// Mitsubishi GX Works2 project: PLC 미니 프로젝트   PLC: Q03UDV

PROGRAM MAIN
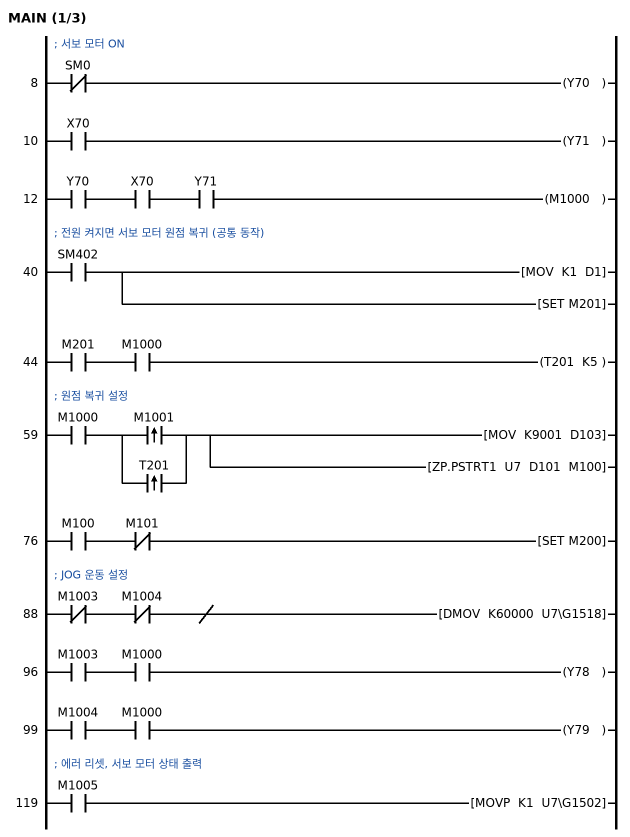
; 서보 모터 ON
8     LDI     SM0
      OUT     Y70
10    LD      X70
      OUT     Y71
12    LD      Y70
      AND     X70
      AND     Y71
      OUT     M1000
; 전원 켜지면 서보 모터 원점 복귀 (공통 동작)
40    LD      SM402
      MOV     K1 D1
      SET     M201
44    LD      M201
      AND     M1000
      OUT     T201 K5
; 원점 복귀 설정
59    LD      M1000
      LDP     M1001
      ORP     T201
      ANB
      MOV     K9001 D103
      ZP.PSTRT1 U7 D101 M100
76    LD      M100
      ANI     M101
      SET     M200
; JOG 운동 설정
88    LDI     M1003
      ANI     M1004
      INV
      DMOV    K60000 U7\G1518
96    LD      M1003
      AND     M1000
      OUT     Y78
99    LD      M1004
      AND     M1000
      OUT     Y79
; 에러 리셋, 서보 모터 상태 출력
119   LD      M1005
      MOVP    K1 U7\G1502
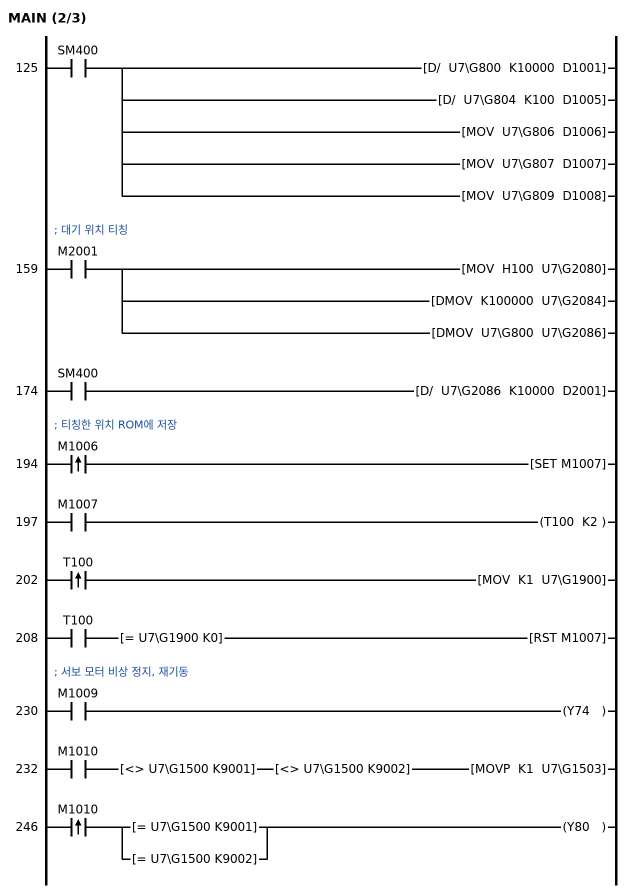
125   LD      SM400
      D/      U7\G800 K10000 D1001
      D/      U7\G804 K100 D1005
      MOV     U7\G806 D1006
      MOV     U7\G807 D1007
      MOV     U7\G809 D1008
; 대기 위치 티칭
159   LD      M2001
      MOV     H100 U7\G2080
      DMOV    K100000 U7\G2084
      DMOV    U7\G800 U7\G2086
174   LD      SM400
      D/      U7\G2086 K10000 D2001
; 티칭한 위치 ROM에 저장
194   LDP     M1006
      SET     M1007
197   LD      M1007
      OUT     T100 K2
202   LDP     T100
      MOV     K1 U7\G1900
208   LD      T100
      AND=    U7\G1900 K0
      RST     M1007
; 서보 모터 비상 정지, 재기동
230   LD      M1009
      OUT     Y74
232   LD      M1010
      AND<>   U7\G1500 K9001
      AND<>   U7\G1500 K9002
      MOVP    K1 U7\G1503
246   LDP     M1010
      LD=     U7\G1500 K9001
      OR=     U7\G1500 K9002
      ANB
      OUT     Y80
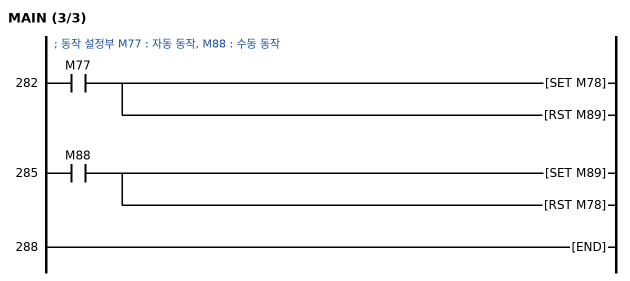
; 동작 설정부 M77 : 자동 동작, M88 : 수동 동작
282   LD      M77
      SET     M78
      RST     M89
285   LD      M88
      SET     M89
      RST     M78
288   END
END_PROGRAM

PROGRAM FacCheck
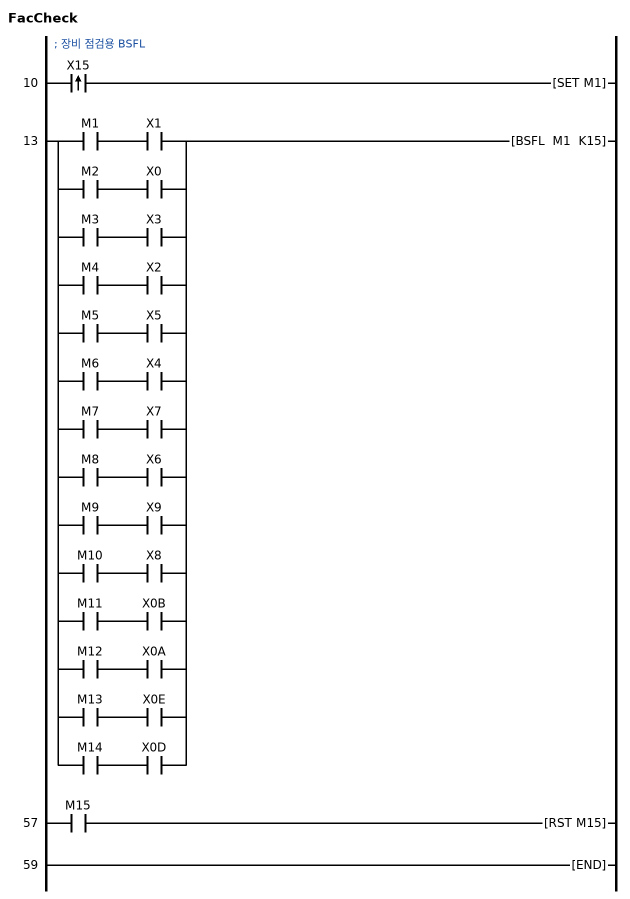
; 장비 점검용 BSFL
10    LDP     X15
      SET     M1
13    LD      M1
      AND     X1
      LD      M2
      AND     X0
      ORB
      LD      M3
      AND     X3
      ORB
      LD      M4
      AND     X2
      ORB
      LD      M5
      AND     X5
      ORB
      LD      M6
      AND     X4
      ORB
      LD      M7
      AND     X7
      ORB
      LD      M8
      AND     X6
      ORB
      LD      M9
      AND     X9
      ORB
      LD      M10
      AND     X8
      ORB
      LD      M11
      AND     X0B
      ORB
      LD      M12
      AND     X0A
      ORB
      LD      M13
      AND     X0E
      ORB
      LD      M14
      AND     X0D
      ORB
      BSFL    M1 K15
57    LD      M15
      RST     M15
59    END
END_PROGRAM

PROGRAM Auto
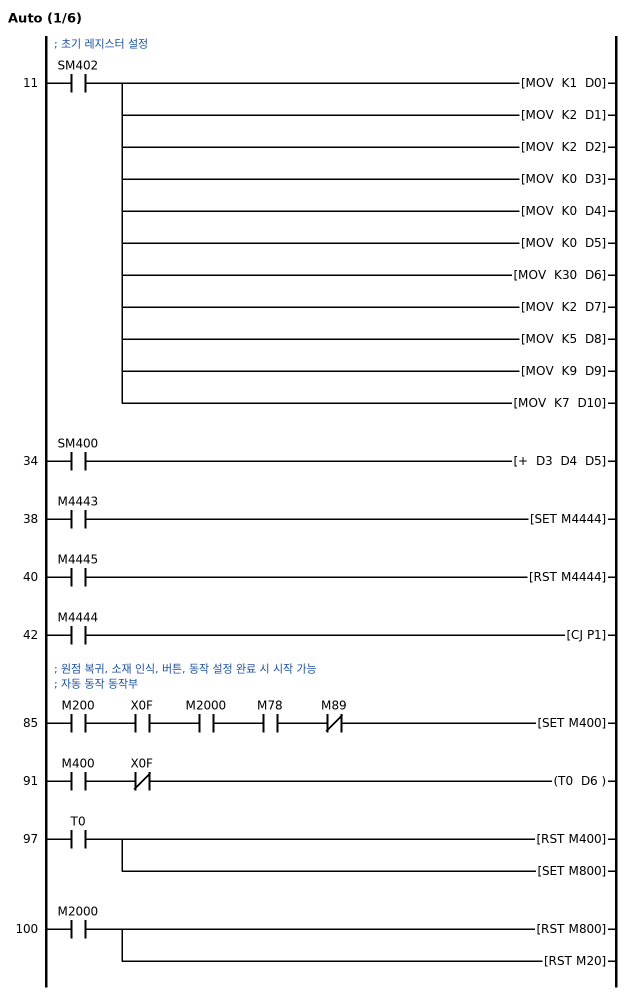
; 초기 레지스터 설정
11    LD      SM402
      MOV     K1 D0
      MOV     K2 D1
      MOV     K2 D2
      MOV     K0 D3
      MOV     K0 D4
      MOV     K0 D5
      MOV     K30 D6
      MOV     K2 D7
      MOV     K5 D8
      MOV     K9 D9
      MOV     K7 D10
34    LD      SM400
      +       D3 D4 D5
38    LD      M4443
      SET     M4444
40    LD      M4445
      RST     M4444
42    LD      M4444
      CJ      P1
; 원점 복귀, 소재 인식, 버튼, 동작 설정 완료 시 시작 가능
; 자동 동작 동작부
85    LD      M200
      AND     X0F
      AND     M2000
      AND     M78
      ANI     M89
      SET     M400
91    LD      M400
      ANI     X0F
      OUT     T0 D6
97    LD      T0
      RST     M400
      SET     M800
100   LD      M2000
      RST     M800
      RST     M20
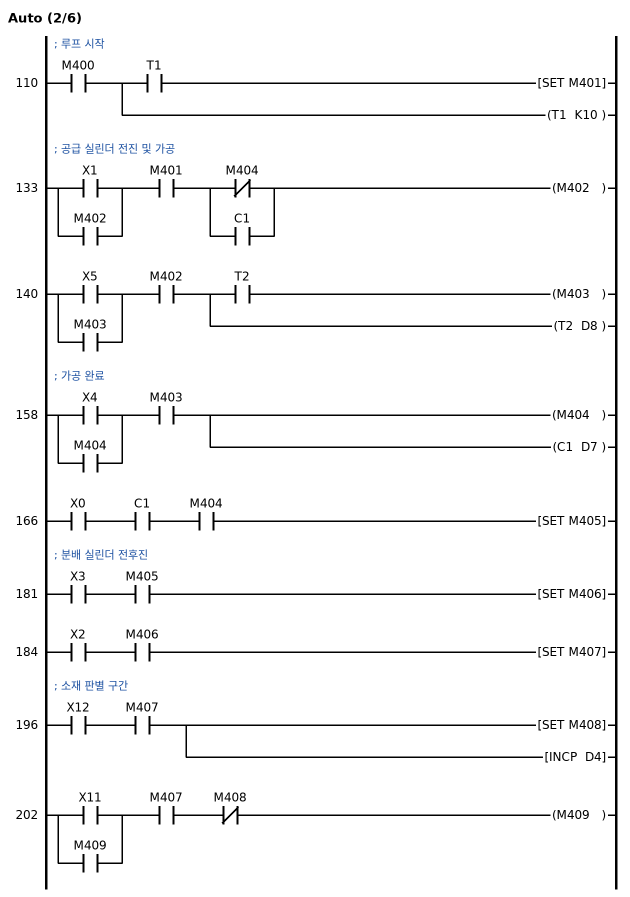
; 루프 시작
110   LD      M400
      MPS
      AND     T1
      SET     M401
      MPP
      OUT     T1 K10
; 공급 실린더 전진 및 가공
133   LD      X1
      OR      M402
      AND     M401
      LDI     M404
      OR      C1
      ANB
      OUT     M402
140   LD      X5
      OR      M403
      AND     M402
      MPS
      AND     T2
      OUT     M403
      MPP
      OUT     T2 D8
; 가공 완료
158   LD      X4
      OR      M404
      AND     M403
      OUT     M404
      OUT     C1 D7
166   LD      X0
      AND     C1
      AND     M404
      SET     M405
; 분배 실린더 전후진
181   LD      X3
      AND     M405
      SET     M406
184   LD      X2
      AND     M406
      SET     M407
; 소재 판별 구간
196   LD      X12
      AND     M407
      SET     M408
      INCP    D4
202   LD      X11
      OR      M409
      AND     M407
      ANI     M408
      OUT     M409
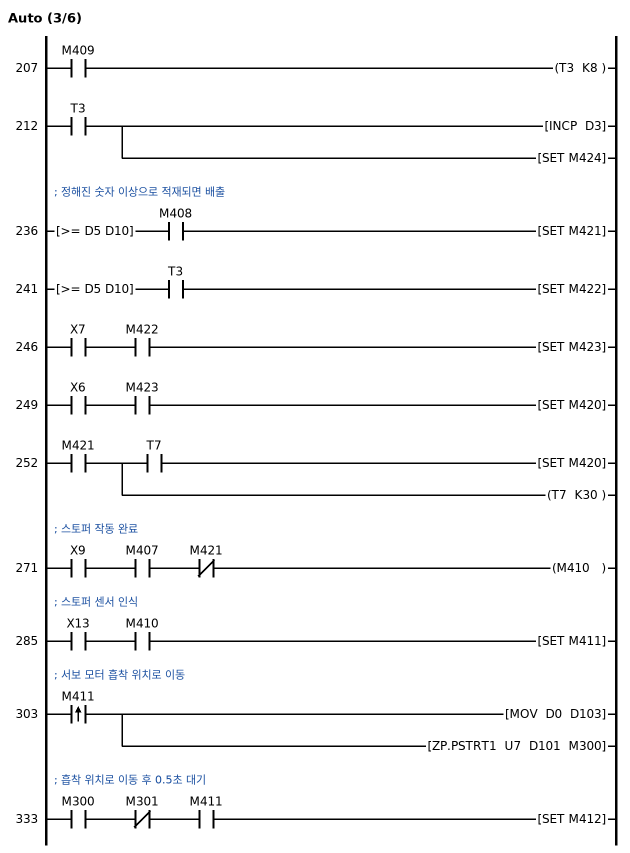
207   LD      M409
      OUT     T3 K8
212   LD      T3
      INCP    D3
      SET     M424
; 정해진 숫자 이상으로 적재되면 배출
236   LD>=    D5 D10
      AND     M408
      SET     M421
241   LD>=    D5 D10
      AND     T3
      SET     M422
246   LD      X7
      AND     M422
      SET     M423
249   LD      X6
      AND     M423
      SET     M420
252   LD      M421
      MPS
      AND     T7
      SET     M420
      MPP
      OUT     T7 K30
; 스토퍼 작동 완료
271   LD      X9
      AND     M407
      ANI     M421
      OUT     M410
; 스토퍼 센서 인식
285   LD      X13
      AND     M410
      SET     M411
; 서보 모터 흡착 위치로 이동
303   LDP     M411
      MOV     D0 D103
      ZP.PSTRT1 U7 D101 M300
; 흡착 위치로 이동 후 0.5초 대기
333   LD      M300
      ANI     M301
      AND     M411
      SET     M412
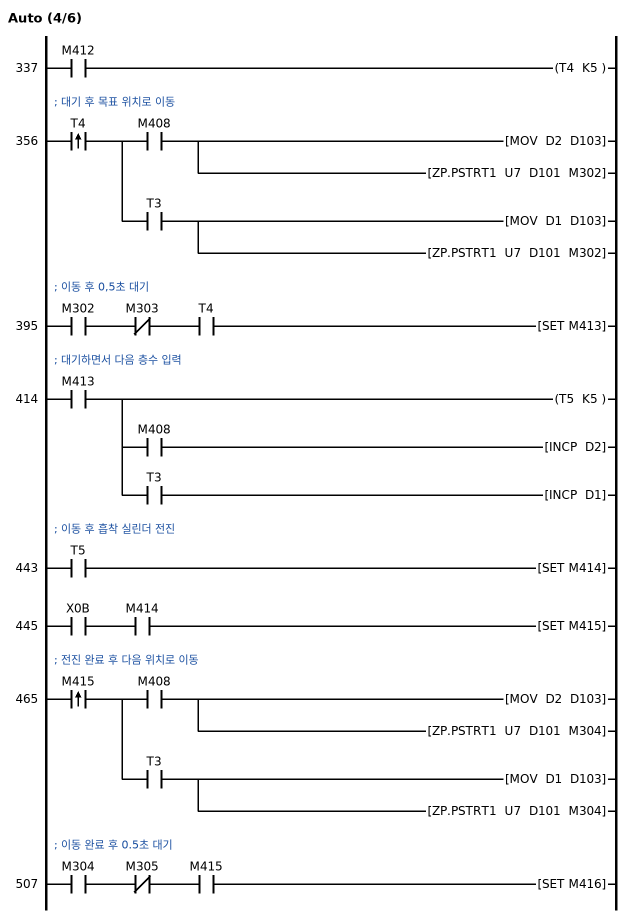
337   LD      M412
      OUT     T4 K5
; 대기 후 목표 위치로 이동
356   LDP     T4
      MPS
      AND     M408
      MOV     D2 D103
      ZP.PSTRT1 U7 D101 M302
      MPP
      AND     T3
      MOV     D1 D103
      ZP.PSTRT1 U7 D101 M302
; 이동 후 0,5초 대기
395   LD      M302
      ANI     M303
      AND     T4
      SET     M413
; 대기하면서 다음 층수 입력
414   LD      M413
      OUT     T5 K5
      MPS
      AND     M408
      INCP    D2
      MPP
      AND     T3
      INCP    D1
; 이동 후 흡착 실린더 전진
443   LD      T5
      SET     M414
445   LD      X0B
      AND     M414
      SET     M415
; 전진 완료 후 다음 위치로 이동
465   LDP     M415
      MPS
      AND     M408
      MOV     D2 D103
      ZP.PSTRT1 U7 D101 M304
      MPP
      AND     T3
      MOV     D1 D103
      ZP.PSTRT1 U7 D101 M304
; 이동 완료 후 0.5초 대기
507   LD      M304
      ANI     M305
      AND     M415
      SET     M416
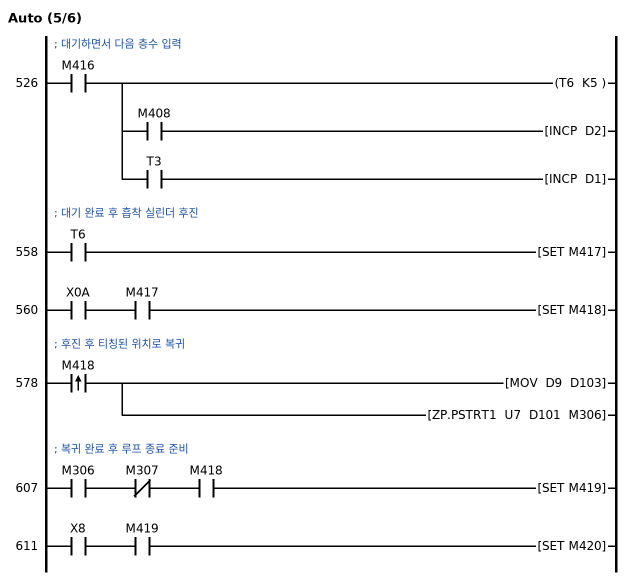
; 대기하면서 다음 층수 입력
526   LD      M416
      OUT     T6 K5
      MPS
      AND     M408
      INCP    D2
      MPP
      AND     T3
      INCP    D1
; 대기 완료 후 흡착 실린더 후진
558   LD      T6
      SET     M417
560   LD      X0A
      AND     M417
      SET     M418
; 후진 후 티칭된 위치로 복귀
578   LDP     M418
      MOV     D9 D103
      ZP.PSTRT1 U7 D101 M306
; 복귀 완료 후 루프 종료 준비
607   LD      M306
      ANI     M307
      AND     M418
      SET     M419
611   LD      X8
      AND     M419
      SET     M420
      P1
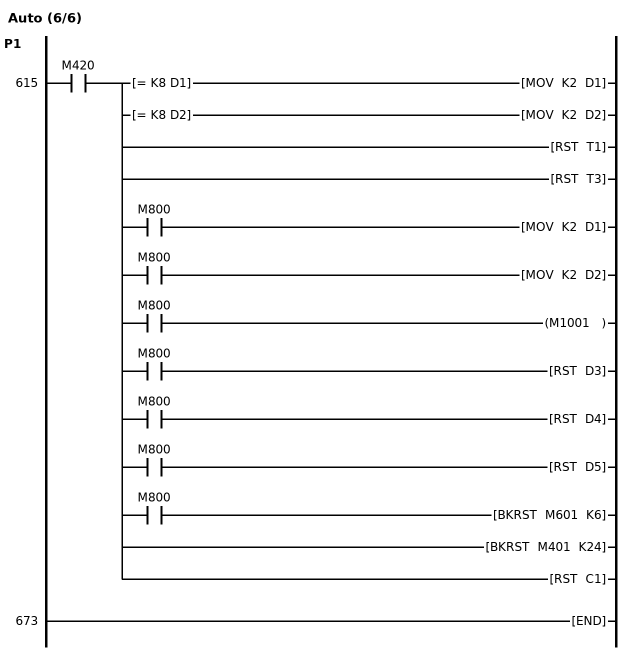
615   LD      M420
      MPS
      AND=    K8 D1
      MOV     K2 D1
      MRD
      AND=    K8 D2
      MOV     K2 D2
      MPP
      RST     T1
      RST     T3
      MPS
      AND     M800
      MOV     K2 D1
      MRD
      AND     M800
      MOV     K2 D2
      MRD
      AND     M800
      OUT     M1001
      MRD
      AND     M800
      RST     D3
      MRD
      AND     M800
      RST     D4
      MRD
      AND     M800
      RST     D5
      MRD
      AND     M800
      BKRST   M601 K6
      MPP
      BKRST   M401 K24
      RST     C1
673   END
END_PROGRAM

PROGRAM Output
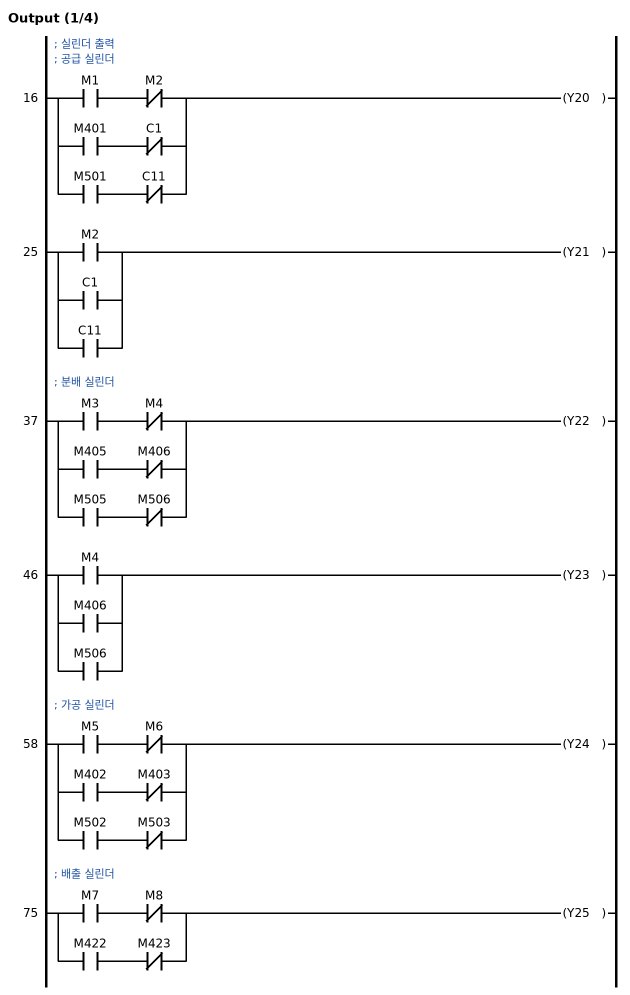
; 실린더 출력
; 공급 실린더
16    LD      M1
      ANI     M2
      LD      M401
      ANI     C1
      ORB
      LD      M501
      ANI     C11
      ORB
      OUT     Y20
25    LD      M2
      OR      C1
      OR      C11
      OUT     Y21
; 분배 실린더
37    LD      M3
      ANI     M4
      LD      M405
      ANI     M406
      ORB
      LD      M505
      ANI     M506
      ORB
      OUT     Y22
46    LD      M4
      OR      M406
      OR      M506
      OUT     Y23
; 가공 실린더
58    LD      M5
      ANI     M6
      LD      M402
      ANI     M403
      ORB
      LD      M502
      ANI     M503
      ORB
      OUT     Y24
; 배출 실린더
75    LD      M7
      ANI     M8
      LD      M422
      ANI     M423
      ORB
      OUT     Y25
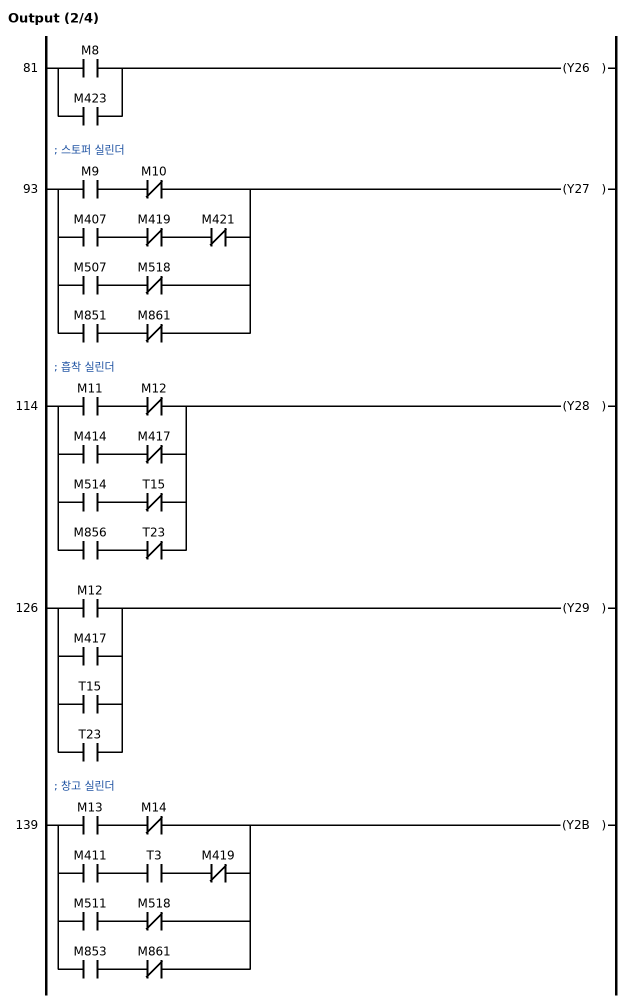
81    LD      M8
      OR      M423
      OUT     Y26
; 스토퍼 실린더
93    LD      M9
      ANI     M10
      LD      M407
      ANI     M419
      ANI     M421
      ORB
      LD      M507
      ANI     M518
      ORB
      LD      M851
      ANI     M861
      ORB
      OUT     Y27
; 흡착 실린더
114   LD      M11
      ANI     M12
      LD      M414
      ANI     M417
      ORB
      LD      M514
      ANI     T15
      ORB
      LD      M856
      ANI     T23
      ORB
      OUT     Y28
126   LD      M12
      OR      M417
      OR      T15
      OR      T23
      OUT     Y29
; 창고 실린더
139   LD      M13
      ANI     M14
      LD      M411
      AND     T3
      ANI     M419
      ORB
      LD      M511
      ANI     M518
      ORB
      LD      M853
      ANI     M861
      ORB
      OUT     Y2B
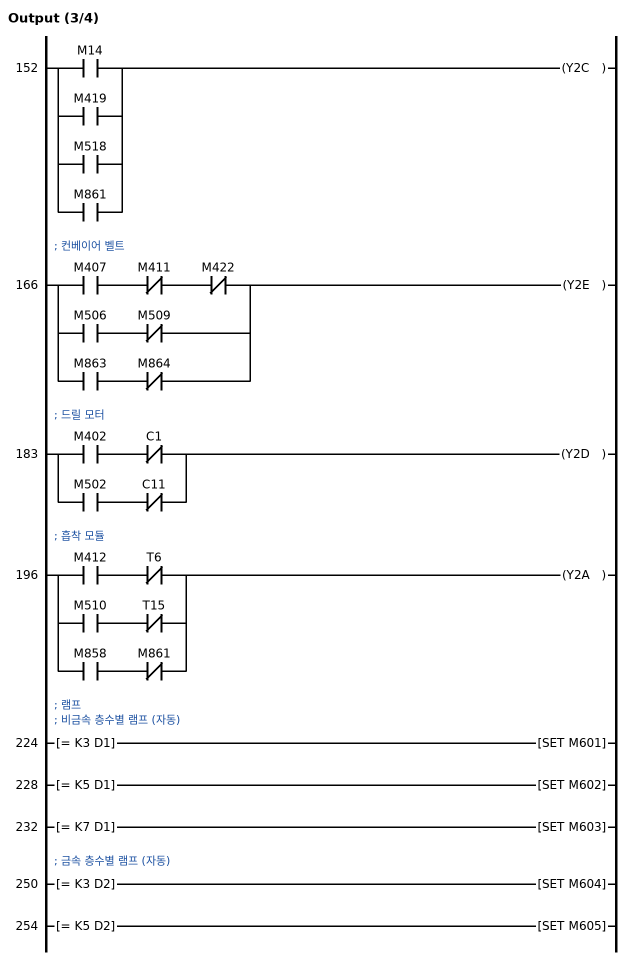
152   LD      M14
      OR      M419
      OR      M518
      OR      M861
      OUT     Y2C
; 컨베이어 벨트
166   LD      M407
      ANI     M411
      ANI     M422
      LD      M506
      ANI     M509
      ORB
      LD      M863
      ANI     M864
      ORB
      OUT     Y2E
; 드릴 모터
183   LD      M402
      ANI     C1
      LD      M502
      ANI     C11
      ORB
      OUT     Y2D
; 흡착 모듈
196   LD      M412
      ANI     T6
      LD      M510
      ANI     T15
      ORB
      LD      M858
      ANI     M861
      ORB
      OUT     Y2A
; 램프
; 비금속 층수별 램프 (자동)
224   LD=     K3 D1
      SET     M601
228   LD=     K5 D1
      SET     M602
232   LD=     K7 D1
      SET     M603
; 금속 층수별 램프 (자동)
250   LD=     K3 D2
      SET     M604
254   LD=     K5 D2
      SET     M605
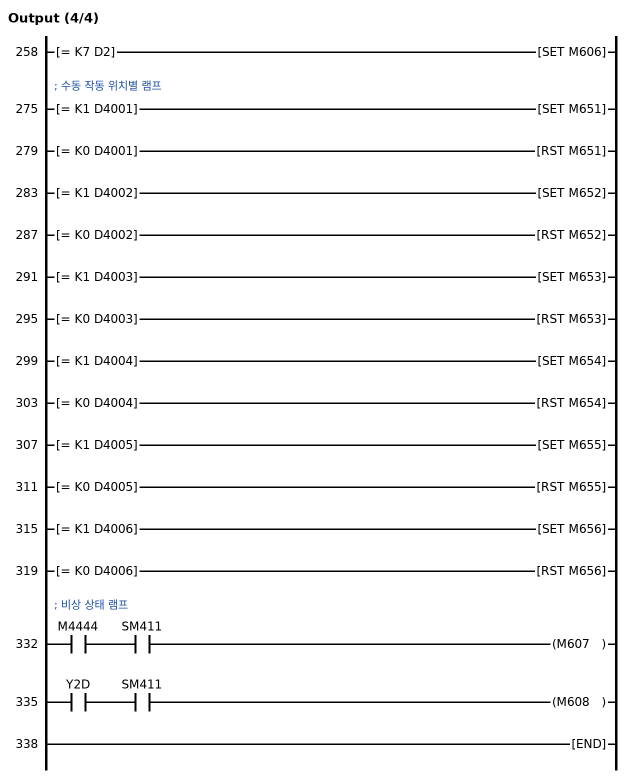
258   LD=     K7 D2
      SET     M606
; 수동 작동 위치별 램프
275   LD=     K1 D4001
      SET     M651
279   LD=     K0 D4001
      RST     M651
283   LD=     K1 D4002
      SET     M652
287   LD=     K0 D4002
      RST     M652
291   LD=     K1 D4003
      SET     M653
295   LD=     K0 D4003
      RST     M653
299   LD=     K1 D4004
      SET     M654
303   LD=     K0 D4004
      RST     M654
307   LD=     K1 D4005
      SET     M655
311   LD=     K0 D4005
      RST     M655
315   LD=     K1 D4006
      SET     M656
319   LD=     K0 D4006
      RST     M656
; 비상 상태 램프
332   LD      M4444
      AND     SM411
      OUT     M607
335   LD      Y2D
      AND     SM411
      OUT     M608
338   END
END_PROGRAM

PROGRAM Manual
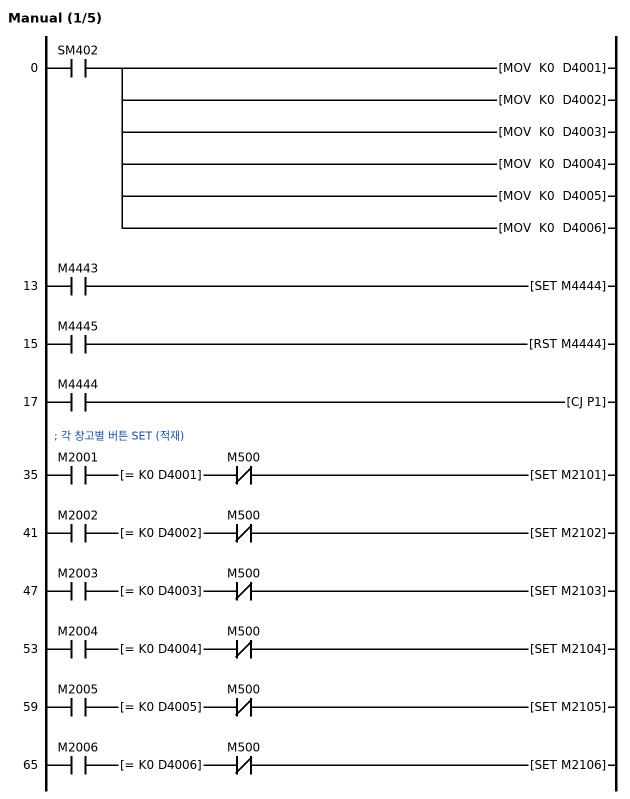
0     LD      SM402
      MOV     K0 D4001
      MOV     K0 D4002
      MOV     K0 D4003
      MOV     K0 D4004
      MOV     K0 D4005
      MOV     K0 D4006
13    LD      M4443
      SET     M4444
15    LD      M4445
      RST     M4444
17    LD      M4444
      CJ      P1
; 각 창고별 버튼 SET (적재)
35    LD      M2001
      AND=    K0 D4001
      ANI     M500
      SET     M2101
41    LD      M2002
      AND=    K0 D4002
      ANI     M500
      SET     M2102
47    LD      M2003
      AND=    K0 D4003
      ANI     M500
      SET     M2103
53    LD      M2004
      AND=    K0 D4004
      ANI     M500
      SET     M2104
59    LD      M2005
      AND=    K0 D4005
      ANI     M500
      SET     M2105
65    LD      M2006
      AND=    K0 D4006
      ANI     M500
      SET     M2106
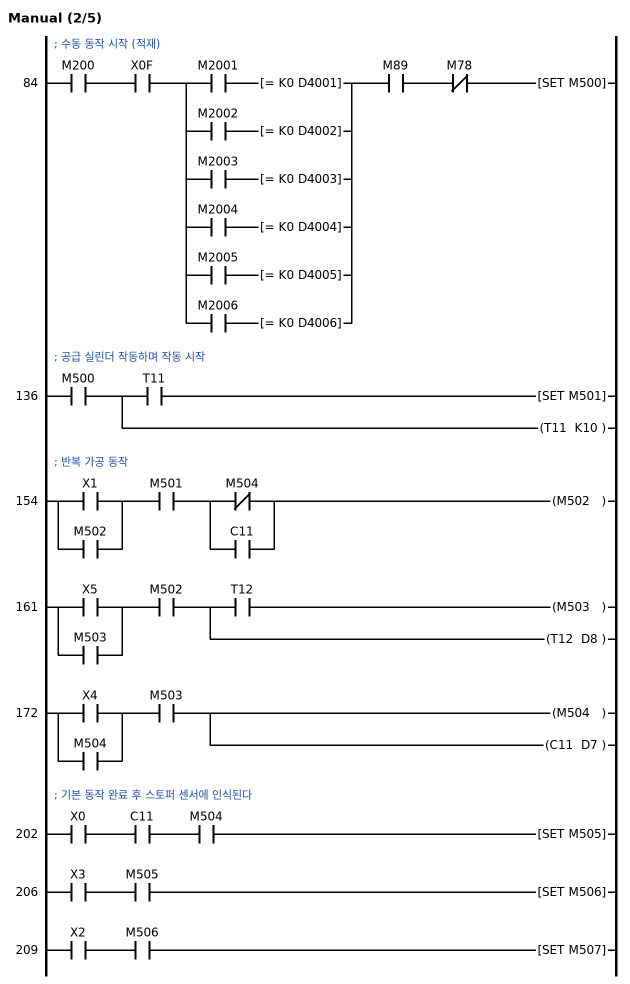
; 수동 동작 시작 (적재)
84    LD      M200
      AND     X0F
      LD      M2001
      AND=    K0 D4001
      LD      M2002
      AND=    K0 D4002
      ORB
      LD      M2003
      AND=    K0 D4003
      ORB
      LD      M2004
      AND=    K0 D4004
      ORB
      LD      M2005
      AND=    K0 D4005
      ORB
      LD      M2006
      AND=    K0 D4006
      ORB
      ANB
      AND     M89
      ANI     M78
      SET     M500
; 공급 실린더 작동하며 작동 시작
136   LD      M500
      MPS
      AND     T11
      SET     M501
      MPP
      OUT     T11 K10
; 반복 가공 동작
154   LD      X1
      OR      M502
      AND     M501
      LDI     M504
      OR      C11
      ANB
      OUT     M502
161   LD      X5
      OR      M503
      AND     M502
      MPS
      AND     T12
      OUT     M503
      MPP
      OUT     T12 D8
172   LD      X4
      OR      M504
      AND     M503
      OUT     M504
      OUT     C11 D7
; 기본 동작 완료 후 스토퍼 센서에 인식된다
202   LD      X0
      AND     C11
      AND     M504
      SET     M505
206   LD      X3
      AND     M505
      SET     M506
209   LD      X2
      AND     M506
      SET     M507
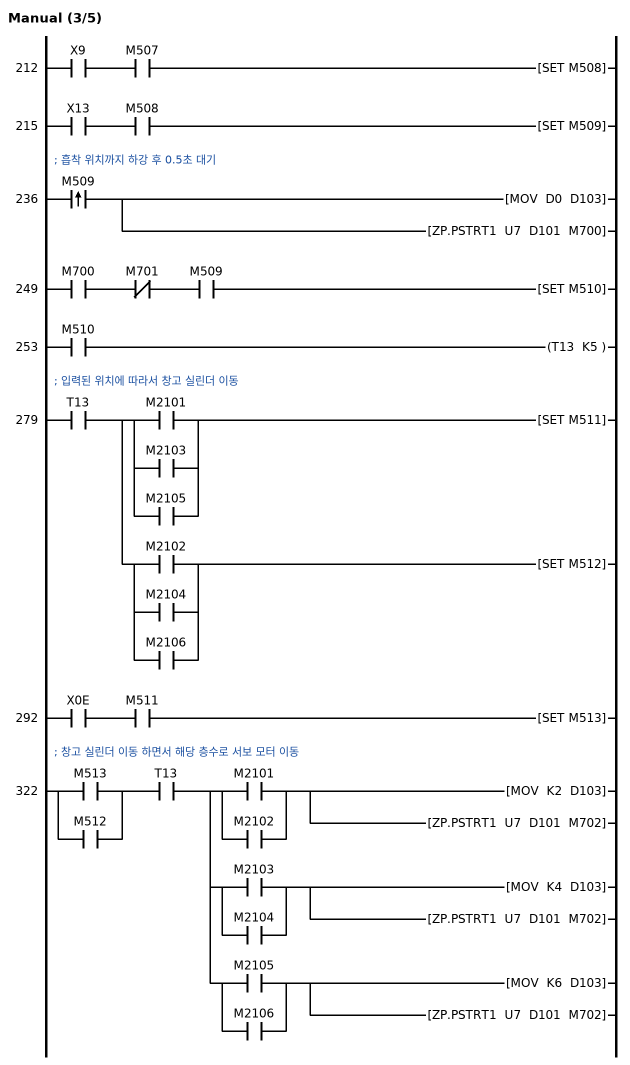
212   LD      X9
      AND     M507
      SET     M508
215   LD      X13
      AND     M508
      SET     M509
; 흡착 위치까지 하강 후 0.5초 대기
236   LDP     M509
      MOV     D0 D103
      ZP.PSTRT1 U7 D101 M700
249   LD      M700
      ANI     M701
      AND     M509
      SET     M510
253   LD      M510
      OUT     T13 K5
; 입력된 위치에 따라서 창고 실린더 이동
279   LD      T13
      MPS
      LD      M2101
      OR      M2103
      OR      M2105
      ANB
      SET     M511
      MPP
      LD      M2102
      OR      M2104
      OR      M2106
      ANB
      SET     M512
292   LD      X0E
      AND     M511
      SET     M513
; 창고 실린더 이동 하면서 해당 층수로 서보 모터 이동
322   LD      M513
      OR      M512
      AND     T13
      MPS
      LD      M2101
      OR      M2102
      ANB
      MOV     K2 D103
      ZP.PSTRT1 U7 D101 M702
      MRD
      LD      M2103
      OR      M2104
      ANB
      MOV     K4 D103
      ZP.PSTRT1 U7 D101 M702
      MPP
      LD      M2105
      OR      M2106
      ANB
      MOV     K6 D103
      ZP.PSTRT1 U7 D101 M702
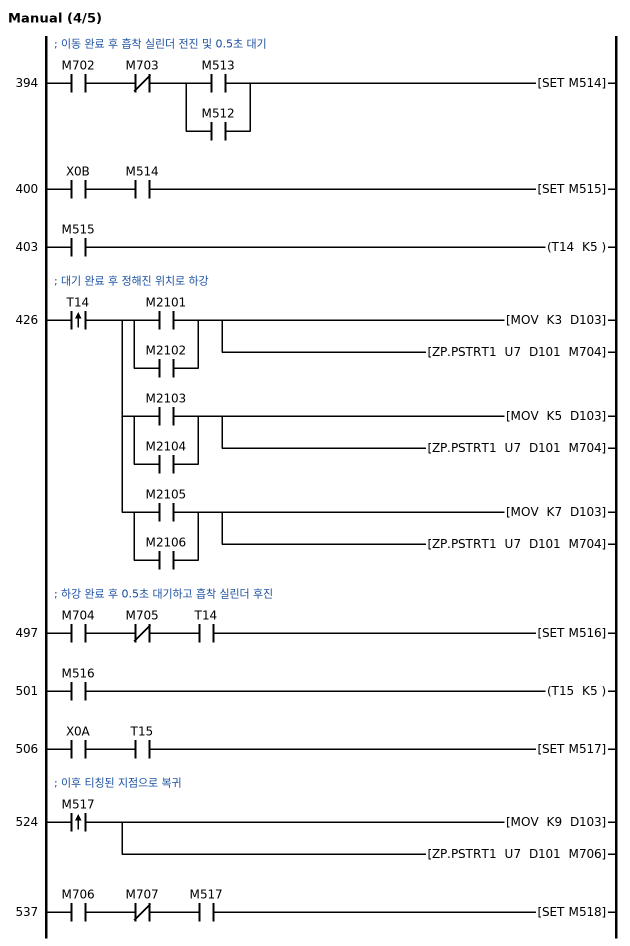
; 이동 완료 후 흡착 실린더 전진 및 0.5초 대기
394   LD      M702
      ANI     M703
      LD      M513
      OR      M512
      ANB
      SET     M514
400   LD      X0B
      AND     M514
      SET     M515
403   LD      M515
      OUT     T14 K5
; 대기 완료 후 정해진 위치로 하강
426   LDP     T14
      MPS
      LD      M2101
      OR      M2102
      ANB
      MOV     K3 D103
      ZP.PSTRT1 U7 D101 M704
      MRD
      LD      M2103
      OR      M2104
      ANB
      MOV     K5 D103
      ZP.PSTRT1 U7 D101 M704
      MPP
      LD      M2105
      OR      M2106
      ANB
      MOV     K7 D103
      ZP.PSTRT1 U7 D101 M704
; 하강 완료 후 0.5초 대기하고 흡착 실린더 후진
497   LD      M704
      ANI     M705
      AND     T14
      SET     M516
501   LD      M516
      OUT     T15 K5
506   LD      X0A
      AND     T15
      SET     M517
; 이후 티칭된 지점으로 복귀
524   LDP     M517
      MOV     K9 D103
      ZP.PSTRT1 U7 D101 M706
537   LD      M706
      ANI     M707
      AND     M517
      SET     M518
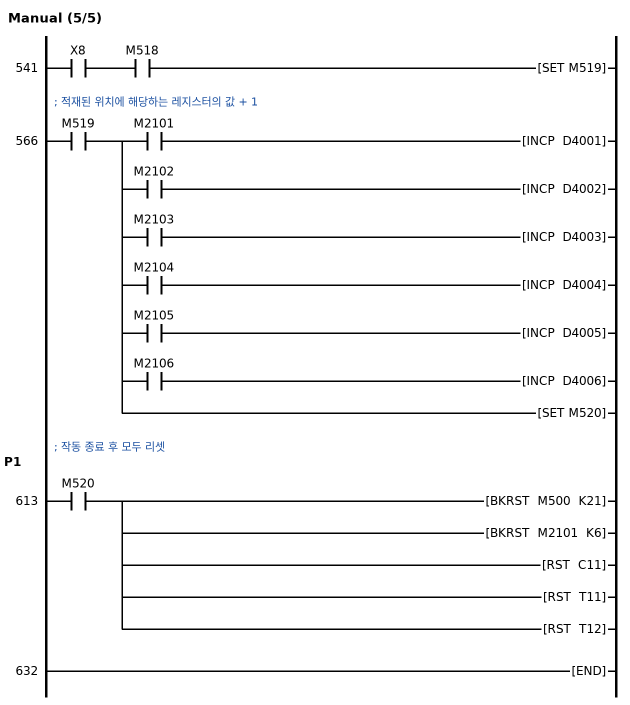
541   LD      X8
      AND     M518
      SET     M519
; 적재된 위치에 해당하는 레지스터의 값 + 1
566   LD      M519
      MPS
      AND     M2101
      INCP    D4001
      MRD
      AND     M2102
      INCP    D4002
      MRD
      AND     M2103
      INCP    D4003
      MRD
      AND     M2104
      INCP    D4004
      MRD
      AND     M2105
      INCP    D4005
      MRD
      AND     M2106
      INCP    D4006
      MPP
      SET     M520
; 작동 종료 후 모두 리셋
      P1
613   LD      M520
      BKRST   M500 K21
      BKRST   M2101 K6
      RST     C11
      RST     T11
      RST     T12
632   END
END_PROGRAM

PROGRAM Manual_2
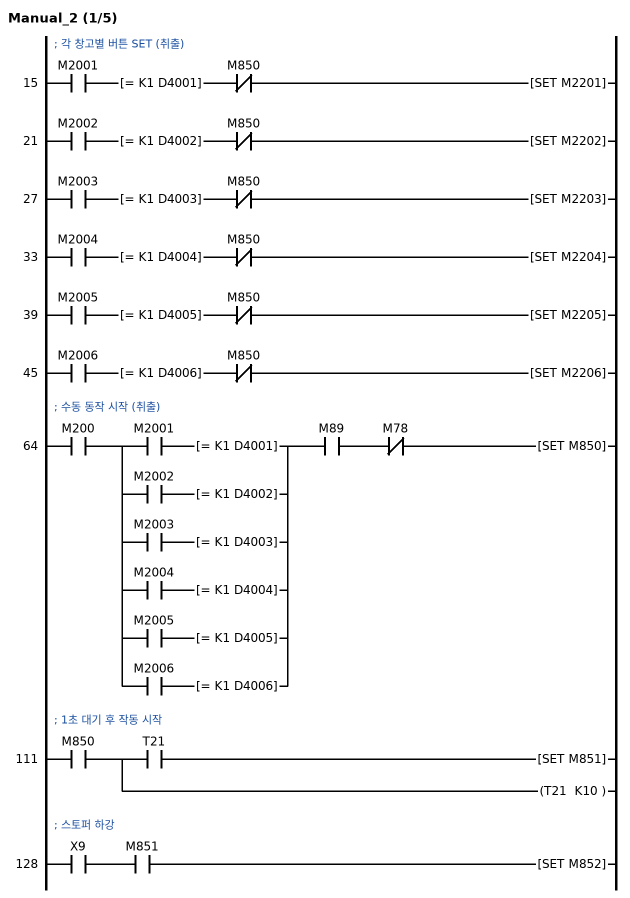
; 각 창고별 버튼 SET (취출)
15    LD      M2001
      AND=    K1 D4001
      ANI     M850
      SET     M2201
21    LD      M2002
      AND=    K1 D4002
      ANI     M850
      SET     M2202
27    LD      M2003
      AND=    K1 D4003
      ANI     M850
      SET     M2203
33    LD      M2004
      AND=    K1 D4004
      ANI     M850
      SET     M2204
39    LD      M2005
      AND=    K1 D4005
      ANI     M850
      SET     M2205
45    LD      M2006
      AND=    K1 D4006
      ANI     M850
      SET     M2206
; 수동 동작 시작 (취출)
64    LD      M200
      LD      M2001
      AND=    K1 D4001
      LD      M2002
      AND=    K1 D4002
      ORB
      LD      M2003
      AND=    K1 D4003
      ORB
      LD      M2004
      AND=    K1 D4004
      ORB
      LD      M2005
      AND=    K1 D4005
      ORB
      LD      M2006
      AND=    K1 D4006
      ORB
      ANB
      AND     M89
      ANI     M78
      SET     M850
; 1초 대기 후 작동 시작
111   LD      M850
      MPS
      AND     T21
      SET     M851
      MPP
      OUT     T21 K10
; 스토퍼 하강
128   LD      X9
      AND     M851
      SET     M852
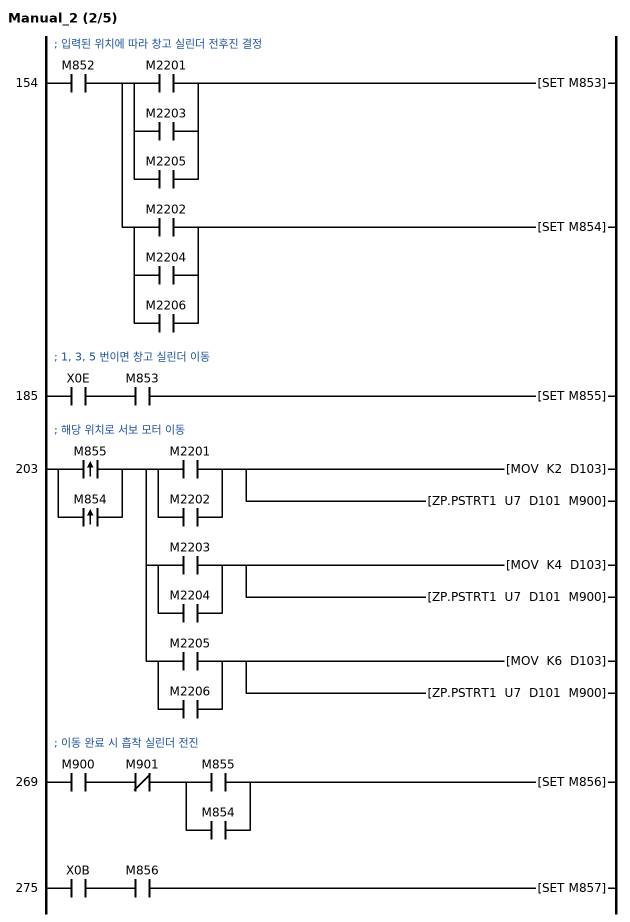
; 입력된 위치에 따라 창고 실린더 전후진 결정
154   LD      M852
      MPS
      LD      M2201
      OR      M2203
      OR      M2205
      ANB
      SET     M853
      MPP
      LD      M2202
      OR      M2204
      OR      M2206
      ANB
      SET     M854
; 1, 3, 5 번이면 창고 실린더 이동
185   LD      X0E
      AND     M853
      SET     M855
; 해당 위치로 서보 모터 이동
203   LDP     M855
      ORP     M854
      MPS
      LD      M2201
      OR      M2202
      ANB
      MOV     K2 D103
      ZP.PSTRT1 U7 D101 M900
      MRD
      LD      M2203
      OR      M2204
      ANB
      MOV     K4 D103
      ZP.PSTRT1 U7 D101 M900
      MPP
      LD      M2205
      OR      M2206
      ANB
      MOV     K6 D103
      ZP.PSTRT1 U7 D101 M900
; 이동 완료 시 흡착 실린더 전진
269   LD      M900
      ANI     M901
      LD      M855
      OR      M854
      ANB
      SET     M856
275   LD      X0B
      AND     M856
      SET     M857
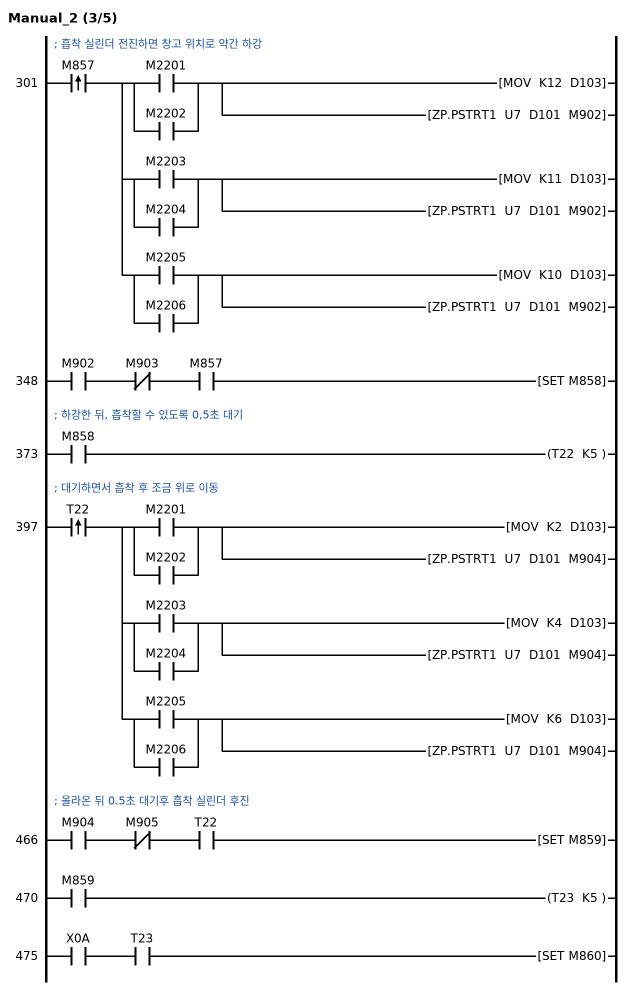
; 흡착 실린더 전진하면 창고 위치로 약간 하강
301   LDP     M857
      MPS
      LD      M2201
      OR      M2202
      ANB
      MOV     K12 D103
      ZP.PSTRT1 U7 D101 M902
      MRD
      LD      M2203
      OR      M2204
      ANB
      MOV     K11 D103
      ZP.PSTRT1 U7 D101 M902
      MPP
      LD      M2205
      OR      M2206
      ANB
      MOV     K10 D103
      ZP.PSTRT1 U7 D101 M902
348   LD      M902
      ANI     M903
      AND     M857
      SET     M858
; 하강한 뒤, 흡착할 수 있도록 0,5초 대기
373   LD      M858
      OUT     T22 K5
; 대기하면서 흡착 후 조금 위로 이동
397   LDP     T22
      MPS
      LD      M2201
      OR      M2202
      ANB
      MOV     K2 D103
      ZP.PSTRT1 U7 D101 M904
      MRD
      LD      M2203
      OR      M2204
      ANB
      MOV     K4 D103
      ZP.PSTRT1 U7 D101 M904
      MPP
      LD      M2205
      OR      M2206
      ANB
      MOV     K6 D103
      ZP.PSTRT1 U7 D101 M904
; 올라온 뒤 0.5초 대기후 흡착 실린더 후진
466   LD      M904
      ANI     M905
      AND     T22
      SET     M859
470   LD      M859
      OUT     T23 K5
475   LD      X0A
      AND     T23
      SET     M860
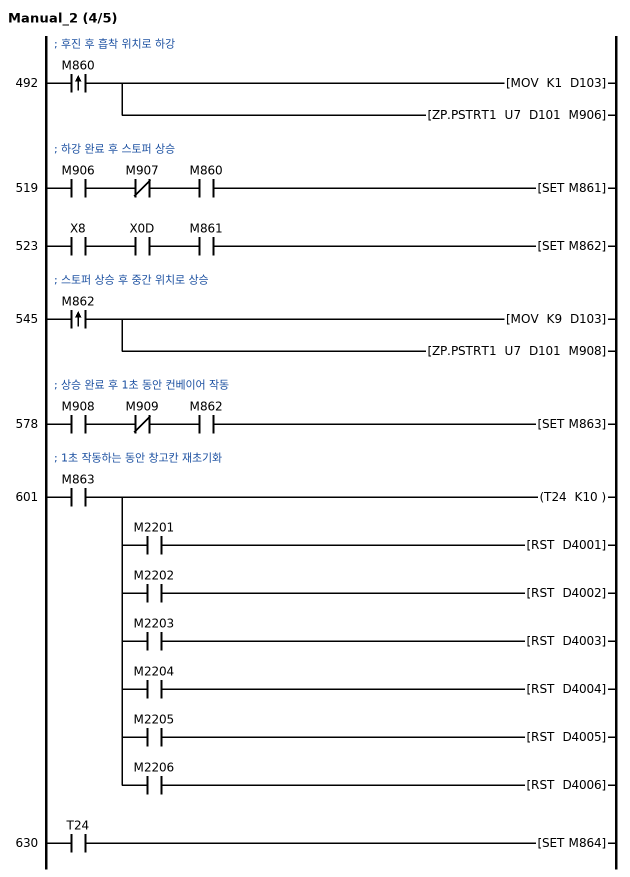
; 후진 후 흡착 위치로 하강
492   LDP     M860
      MOV     K1 D103
      ZP.PSTRT1 U7 D101 M906
; 하강 완료 후 스토퍼 상승
519   LD      M906
      ANI     M907
      AND     M860
      SET     M861
523   LD      X8
      AND     X0D
      AND     M861
      SET     M862
; 스토퍼 상승 후 중간 위치로 상승
545   LDP     M862
      MOV     K9 D103
      ZP.PSTRT1 U7 D101 M908
; 상승 완료 후 1초 동안 컨베이어 작동
578   LD      M908
      ANI     M909
      AND     M862
      SET     M863
; 1초 작동하는 동안 창고칸 재초기화
601   LD      M863
      OUT     T24 K10
      MPS
      AND     M2201
      RST     D4001
      MRD
      AND     M2202
      RST     D4002
      MRD
      AND     M2203
      RST     D4003
      MRD
      AND     M2204
      RST     D4004
      MRD
      AND     M2205
      RST     D4005
      MPP
      AND     M2206
      RST     D4006
630   LD      T24
      SET     M864
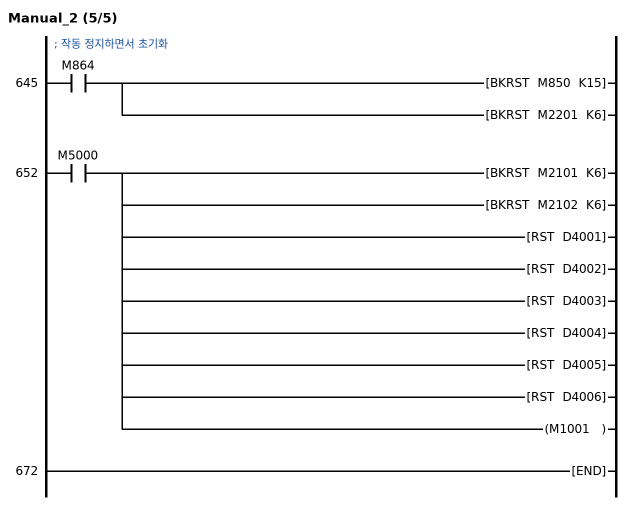
; 작동 정지하면서 초기화
645   LD      M864
      BKRST   M850 K15
      BKRST   M2201 K6
652   LD      M5000
      BKRST   M2101 K6
      BKRST   M2102 K6
      RST     D4001
      RST     D4002
      RST     D4003
      RST     D4004
      RST     D4005
      RST     D4006
      OUT     M1001
672   END
END_PROGRAM
